GLOBALCONSTANTS AID_FA_FONT (* Font attributes object attribute ids *)
  (* Standard: 61499-1; Description: Copyright (c) 2023 HR Agrartechnik GmbH This program and the accompanying materials are made available under the terms of the Eclipse Public License 2.0 which is available at https://www.eclipse.org/legal/epl-2.0/ SPDX-License-Identifier: EPL-2.0 *)
  (* Version 1.0, 2026-06-20, Franz Höpfinger, HR Agrartechnik GmbH *)
  PACKAGE isobus::UT::Q::const::AID;
  IMPORT eclipse4diac::core::TypeHash;
  VAR_GLOBAL CONSTANT
    COLOUR : USINT := USINT#1; (* 1: AID_FA_FONT_COLOUR - Colour index. *)
    SIZE : USINT := USINT#2; (* 2: AID_FA_FONT_SIZE *)
    FONT_TYPE : USINT := USINT#3; (* 3: AID_FA_FONT_FONT_TYPE *)
    STYLE : USINT := USINT#4; (* 4: AID_FA_FONT_STYLE - Bitmask: Bit 0=Bold, Bit 1=Crossed Out, Bit 2=Underlined, Bit 3=Italic, Bit 4=Inverted, Bit 5=Flashing inverted, Bit 6=Flashing hidden, Bit 7=Proportional rendering. *)
  END_VAR
END_GLOBALCONSTANTS
